(* PLC project TreuilsBenneStaging.project, CODESYS CODESYS V3.5 SP19 Patch 1 *)
(* stored: creationDateTime 2026-08-02T00:00:00, modificationDateTime 2026-08-02T00:00:00 *)

PROGRAM PRG_04_Treuils_Benne_CFC
  VAR_OUTPUT
    M1SafeStop : BOOL;
    M1PowerCutOff : BOOL;
    M2SafeStop : BOOL;
    M2PowerCutOff : BOOL;
  END_VAR
  VAR
    instTreuilsBenneProjection : FB_TreuilsBenneStagingProjection;
    instSafetyWinchM1 : FB_Safety_Winch;
    instSafetyWinchM2 : FB_Safety_Winch;
    instWinchM1 : FB_Winch;
    instWinchM2 : FB_Winch;
  END_VAR

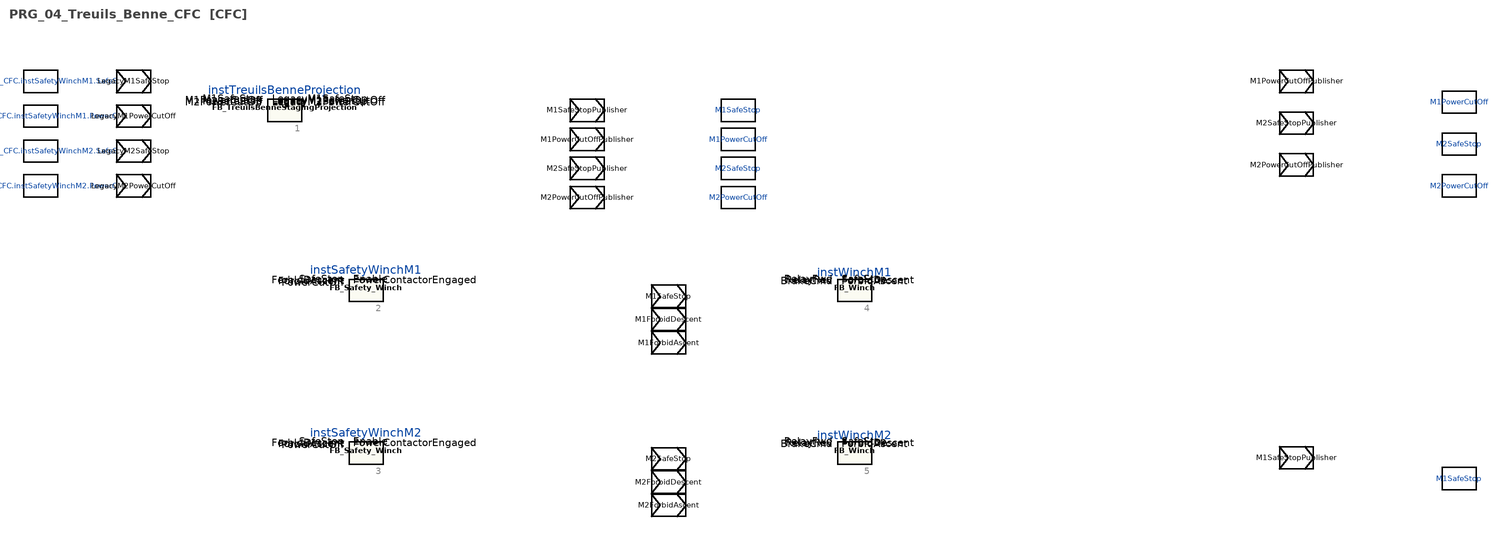
(* CFC diagram, written out as Structured Text *)
instTreuilsBenneProjection(LegacyM1SafeStop := PRG_SAFETY_CFC.instSafetyWinchM1.SafeStop, LegacyM1PowerCutOff := PRG_SAFETY_CFC.instSafetyWinchM1.PowerCutOff, LegacyM2SafeStop := PRG_SAFETY_CFC.instSafetyWinchM2.SafeStop, LegacyM2PowerCutOff := PRG_SAFETY_CFC.instSafetyWinchM2.PowerCutOff);
instSafetyWinchM1(Enable := PRG_SAFETY_CFC.instSafetyWinchM1.SafeStop, PowerContactorEngaged := PRG_SAFETY_CFC.instSafetyWinchM1.PowerCutOff);
instSafetyWinchM2(Enable := PRG_SAFETY_CFC.instSafetyWinchM2.SafeStop, PowerContactorEngaged := PRG_SAFETY_CFC.instSafetyWinchM2.PowerCutOff);
instWinchM1(SafeStop := instSafetyWinchM1.SafeStop, ForbidDescent := instSafetyWinchM1.ForbidDescent, ForbidAscent := instSafetyWinchM1.ForbidAscent);
instWinchM2(SafeStop := instSafetyWinchM2.SafeStop, ForbidDescent := instSafetyWinchM2.ForbidDescent, ForbidAscent := instSafetyWinchM2.ForbidAscent);
M1SafeStop := instTreuilsBenneProjection.M1SafeStop;
M1PowerCutOff := instSafetyWinchM1.PowerCutOff;
M1PowerCutOff := instTreuilsBenneProjection.M1PowerCutOff;
M2SafeStop := instSafetyWinchM2.SafeStop;
M2SafeStop := instTreuilsBenneProjection.M2SafeStop;
M2PowerCutOff := instSafetyWinchM2.PowerCutOff;
M2PowerCutOff := instTreuilsBenneProjection.M2PowerCutOff;
M1SafeStop := instSafetyWinchM1.SafeStop;
END_PROGRAM
